PROGRAM Condition
VAR
	nMark : INT := 88;
	sGrade : STRING ;
END_VAR

ACT_Case();

ACTION ACT_Case:
CASE nMark OF
	 91..100:
	sGrade := 'A';
	81..90 :
	sGrade:= 'B';
	71..80:
	sGrade:= 'C';
	61..70:
	sGrade:= 'D';
	ELSE
		sGrade:= 'F';
	
END_CASE
END_ACTION

ACTION ACT_Condition:
IF nMark > 90 THEN
	sGrade := 'A';
	ELSIF nMark > 80 THEN
		IF nMark > 85 THEN
			sGrade := 'B+';
		ELSE
			sGrade := 'B';
		END_IF
	ELSIF nMark > 70 THEN
		sGrade := 'C';
	ELSIF nMark > 60 THEN
		sGrade := 'D';
	ELSE sGrade := 'F';
END_IF
END_ACTION

END_PROGRAM

(* stored: Version 1.1.0.1, ProductVersion 3.1.4024.16
   POU Condition: Id {fed83c72-9534-4b6f-9d43-f1c5a6d7568e}, SpecialFunc None
   Action ACT_Case: Id {0a815743-c058-4e7f-88c5-956f4f75e7d1}
   Action ACT_Condition: Id {5ee9241c-1e79-49cd-834a-835364c5e10f} *)
